(* Logix 5000 project; controller ProyectoAPMV1 vendor 1 type 14 code 156 rev 30.11; software revision 30.00 *)

TASK MainTask (continuous, watchdog 500 ms) : MainProgram

MODULES
   Local : vendor 1 type 14 code 156 (Compact 0, rev 30.11)
      DCINPUT : 1769-IQ16 (Compact 4, rev 1.1, Input RPI 20 ms)
      DCACOUTPUT : vendor 1 type 7 code 86 (Compact 5, rev 2.1, Output RPI 20 ms)
END_MODULES

VAR_GLOBAL   (* controller tags *)
   Bloquear_Puertas_Horno : BOOL;
   Buffer_Adhesivos : COUNTER := (PRE := 8);
   Buffer_Almacen : COUNTER := (PRE := 1000);
   Buffer_Calidad : COUNTER := (PRE := 8);
   Buffer_Corte : COUNTER := (PRE := 8);
   Buffer_CorteDINT : DINT;
   Buffer_Doblado : COUNTER := (PRE := 8);
   Buffer_Embalaje : COUNTER := (PRE := 100);
   Buffer_Horneado : COUNTER;
   Buffer_Pintado : COUNTER := (PRE := 100);
   Buffer_Pulido : COUNTER := (PRE := 8);
   C0 : BOOL;
   C10 : BOOL;
   C30 : BOOL;
   Contador_Calidad : COUNTER := (PRE := 100);
   E0 : BOOL;   // INICIALIZACION
   E10 : BOOL;
   E100 : BOOL;
   E110 : BOOL;
   E120 : BOOL;
   E130 : BOOL;
   E140 : BOOL;
   E150 : BOOL;
   E160 : BOOL;
   E170 : BOOL;
   E180 : BOOL;
   E190 : BOOL;
   E195 : BOOL;
   E20 : BOOL;
   E200 : BOOL;
   E210 : BOOL;
   E215 : BOOL;
   E220 : BOOL;
   E225 : BOOL;
   E230 : BOOL;
   E235 : BOOL;
   E240 : BOOL;
   E245 : BOOL;
   E250 : BOOL;
   E255 : BOOL;
   E260 : BOOL;
   E270 : BOOL;
   E280 : BOOL;
   E290 : BOOL;
   E30 : BOOL;
   E300 : BOOL;
   E310 : BOOL;
   E330 : BOOL;
   E340 : BOOL;
   E350 : BOOL;
   E360 : BOOL;
   E370 : BOOL;
   E380 : BOOL;
   E390 : BOOL;
   E40 : BOOL;
   E400 : BOOL;
   E410 : BOOL;
   E420 : BOOL;
   E430 : BOOL;
   E440 : BOOL;
   E450 : BOOL;
   E460 : BOOL;
   E50 : BOOL;
   E60 : BOOL;
   E70 : BOOL;
   E80 : BOOL;
   E90 : BOOL;
   Highlighter : BOOL;
   Lote_Piezas : DINT;
   Nro_Laminas : COUNTER := (PRE := 100);
   Parada_Pintado : BOOL;
   Piezas_Almacen : COUNTER := (PRE := 100);
   Pintado1_OK : BOOL;
   Pintado2_OK : BOOL;
   Pintado3_OK : BOOL;
   PlanseSensor2 : BOOL;
   PlanseSensor3 : BOOL;
   PlanseSensor4 : BOOL;
   Pos1ManipuladorOK : BOOL;
   Pos2ManipuladorOK : BOOL;
   Pos3ManipuladorOK : BOOL;
   Puerta_Cabina_Cerrada : BOOL;
   REINICIO_BANDERAS : BOOL;
   SCADA_Piezas : BOOL;
   Sensor_Puertas_Horno : BOOL;
   SimulationStarted : BOOL;
   Start_Adhesivos : BOOL;
   START_ALL : ALIAS FOR Local:4:I.Data.0;
   Start_Lavado : BOOL;
   Start_Pintado : BOOL;
   Start_Pulido : BOOL;
   STOP_ALL : ALIAS FOR Local:4:I.Data.1;
   Timer_Adhesivos : TIMER := (PRE := 10000);
   Timer_Alist_Adhesivos : TIMER := (PRE := 10000);
   Timer_Alist_Corte : TIMER := (PRE := 10000);
   Timer_Alist_Doblado : TIMER := (PRE := 10000);
   Timer_Alist_Embalaje : TIMER := (PRE := 10000);
   Timer_Alist_Horneado : TIMER;
   Timer_Alist_Pintado : TIMER;
   Timer_Alist_Pulido : TIMER := (PRE := 10000);
   Timer_Clasifiacion : TIMER := (PRE := 10000);
   Timer_Corte : TIMER := (PRE := 10000);
   Timer_Despacho : TIMER := (PRE := 1000);
   Timer_Doblado : TIMER := (PRE := 10000);
   Timer_Embalaje : TIMER := (PRE := 10000);
   Timer_Horneado : TIMER := (PRE := 10000);
   Timer_Lavado : TIMER := (PRE := 10000);
   Timer_Pulido : TIMER := (PRE := 10000);
   Timer_Revision_Calidad : TIMER := (PRE := 10000);
   Timer_Transp_Adhesivos : TIMER := (PRE := 10000);
   Timer_Transp_Calidad : TIMER := (PRE := 10000);
   Timer_Transp_Corte : TIMER := (PRE := 10000);
   Timer_Transp_Doblado : TIMER := (PRE := 10000);
   Timer_Transp_Embalaje : TIMER := (PRE := 10000);
   Timer_Transp_Horneado : TIMER := (PRE := 10000);
   Timer_Transp_Lavado : TIMER := (PRE := 10000);
   Timer_Transp_Pintado : TIMER;
   Timer_Transp_Pulido : TIMER := (PRE := 10000);
   Timer_Vac_Horneado : TIMER := (PRE := 1000);
END_VAR

PROGRAM MainProgram   (* main routine MainRoutine *)

ROUTINE Adhesivos   (* ladder *)
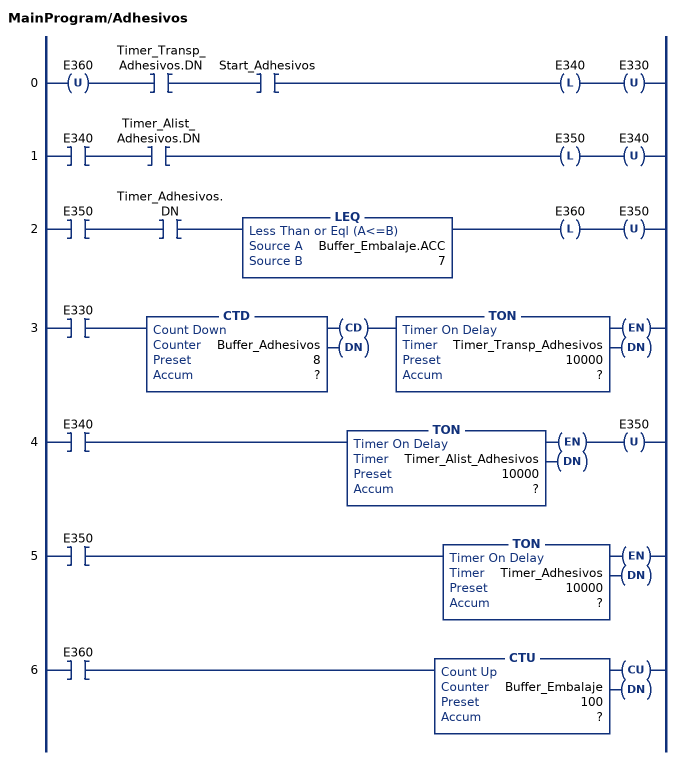
   0: OTU(E360)XIC(Timer_Transp_Adhesivos.DN)XIC(Start_Adhesivos)OTL(E340)OTU(E330);
   1: XIC(E340)XIC(Timer_Alist_Adhesivos.DN)OTL(E350)OTU(E340);
   2: XIC(E350)XIC(Timer_Adhesivos.DN)LEQ(Buffer_Embalaje.ACC,7)OTL(E360)OTU(E350);
   3: XIC(E330)CTD(Buffer_Adhesivos,?,?)TON(Timer_Transp_Adhesivos,?,?);
   4: XIC(E340)TON(Timer_Alist_Adhesivos,?,?)OTU(E350);
   5: XIC(E350)TON(Timer_Adhesivos,?,?);
   6: XIC(E360)CTU(Buffer_Embalaje,?,?);
END_ROUTINE

ROUTINE Almacen   (* ladder *)
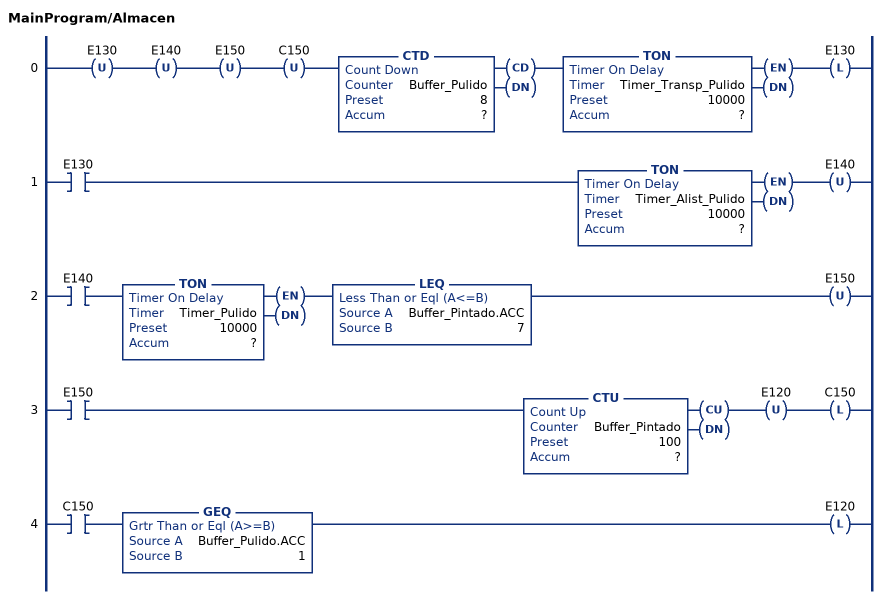
   0: OTU(E130)OTU(E140)OTU(E150)OTU(C150)CTD(Buffer_Pulido,?,?)TON(Timer_Transp_Pulido,?,?)OTL(E130);
   1: XIC(E130)TON(Timer_Alist_Pulido,?,?)OTU(E140);
   2: XIC(E140)TON(Timer_Pulido,?,?)LEQ(Buffer_Pintado.ACC,7)OTU(E150);
   3: XIC(E150)CTU(Buffer_Pintado,?,?)OTU(E120)OTL(C150);
   4: XIC(C150)GEQ(Buffer_Pulido.ACC,1)OTL(E120);
END_ROUTINE

ROUTINE Calidad   (* ladder *)
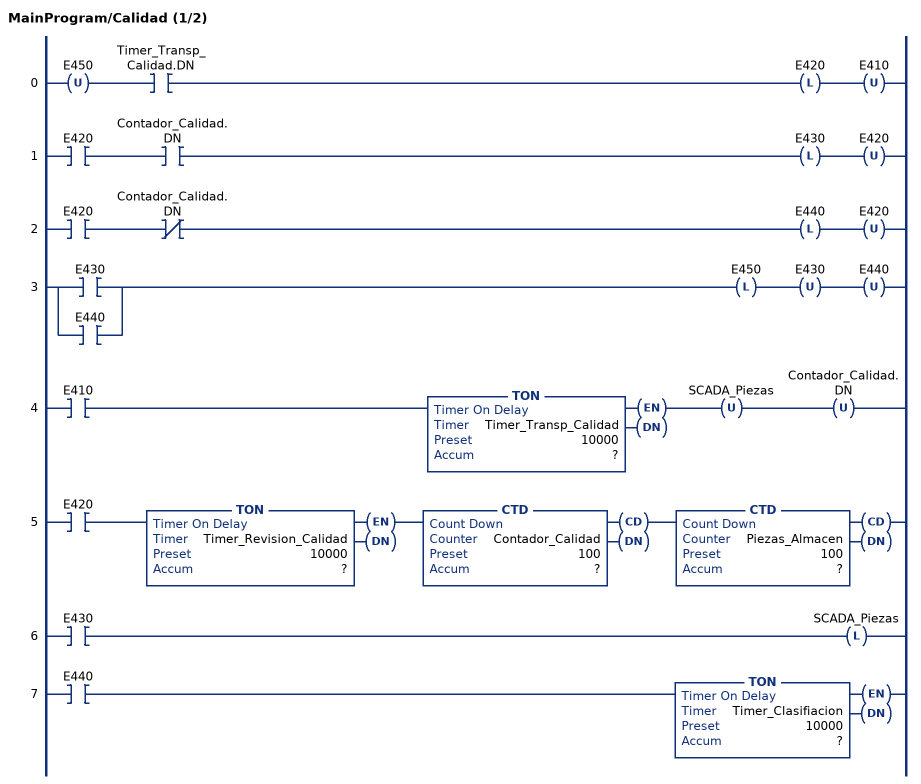
   0: OTU(E450)XIC(Timer_Transp_Calidad.DN)OTL(E420)OTU(E410);
   1: XIC(E420)XIC(Contador_Calidad.DN)OTL(E430)OTU(E420);
   2: XIC(E420)XIO(Contador_Calidad.DN)OTL(E440)OTU(E420);
   3: [XIC(E430) ,XIC(E440) ]OTL(E450)OTU(E430)OTU(E440);
   4: XIC(E410)TON(Timer_Transp_Calidad,?,?)OTU(SCADA_Piezas)OTU(Contador_Calidad.DN);
   5: XIC(E420)TON(Timer_Revision_Calidad,?,?)CTD(Contador_Calidad,?,?)CTD(Piezas_Almacen,?,?);
   6: XIC(E430)OTL(SCADA_Piezas);
   7: XIC(E440)TON(Timer_Clasifiacion,?,?);
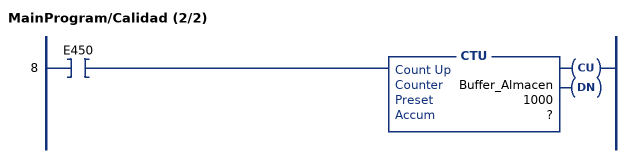
   8: XIC(E450)CTU(Buffer_Almacen,?,?);
END_ROUTINE

ROUTINE Corte_Laminas   (* ladder *)
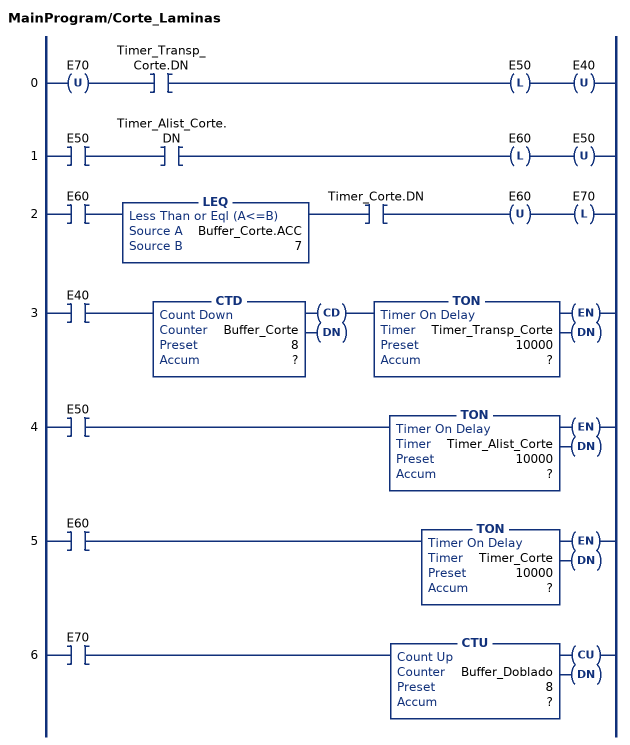
   0: OTU(E70)XIC(Timer_Transp_Corte.DN)OTL(E50)OTU(E40);
   1: XIC(E50)XIC(Timer_Alist_Corte.DN)OTL(E60)OTU(E50);
   2: XIC(E60)LEQ(Buffer_Corte.ACC,7)XIC(Timer_Corte.DN)OTU(E60)OTL(E70);
   3: XIC(E40)CTD(Buffer_Corte,?,?)TON(Timer_Transp_Corte,?,?);
   4: XIC(E50)TON(Timer_Alist_Corte,?,?);
   5: XIC(E60)TON(Timer_Corte,?,?);
   6: XIC(E70)CTU(Buffer_Doblado,?,?);
END_ROUTINE

ROUTINE Doblado_Laminas   (* ladder *)
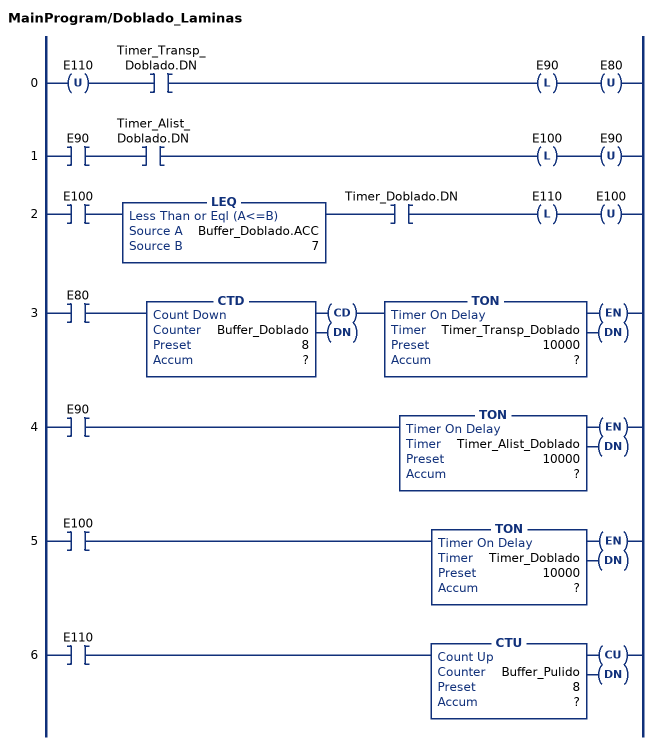
   0: OTU(E110)XIC(Timer_Transp_Doblado.DN)OTL(E90)OTU(E80);
   1: XIC(E90)XIC(Timer_Alist_Doblado.DN)OTL(E100)OTU(E90);
   2: XIC(E100)LEQ(Buffer_Doblado.ACC,7)XIC(Timer_Doblado.DN)OTL(E110)OTU(E100);
   3: XIC(E80)CTD(Buffer_Doblado,?,?)TON(Timer_Transp_Doblado,?,?);
   4: XIC(E90)TON(Timer_Alist_Doblado,?,?);
   5: XIC(E100)TON(Timer_Doblado,?,?);
   6: XIC(E110)CTU(Buffer_Pulido,?,?);
END_ROUTINE

ROUTINE Embalaje   (* ladder *)
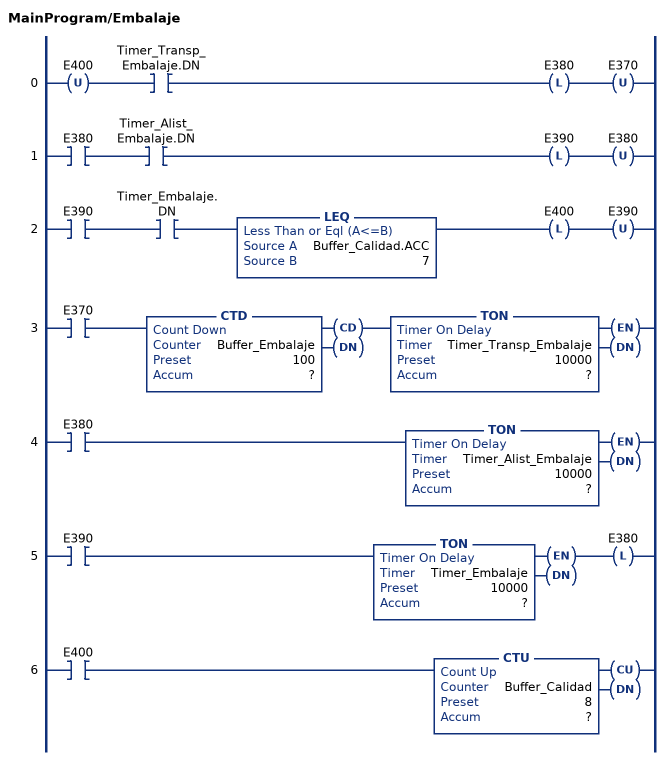
   0: OTU(E400)XIC(Timer_Transp_Embalaje.DN)OTL(E380)OTU(E370);
   1: XIC(E380)XIC(Timer_Alist_Embalaje.DN)OTL(E390)OTU(E380);
   2: XIC(E390)XIC(Timer_Embalaje.DN)LEQ(Buffer_Calidad.ACC,7)OTL(E400)OTU(E390);
   3: XIC(E370)CTD(Buffer_Embalaje,?,?)TON(Timer_Transp_Embalaje,?,?);
   4: XIC(E380)TON(Timer_Alist_Embalaje,?,?);
   5: XIC(E390)TON(Timer_Embalaje,?,?)OTL(E380);
   6: XIC(E400)CTU(Buffer_Calidad,?,?);
END_ROUTINE

ROUTINE Horneado_Piezas   (* ladder *)
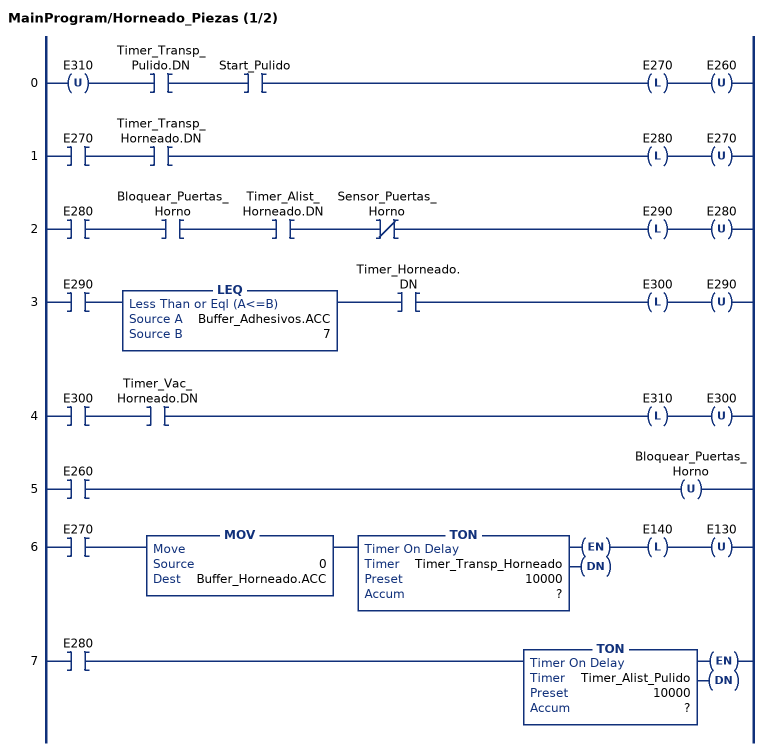
   0: OTU(E310)XIC(Timer_Transp_Pulido.DN)XIC(Start_Pulido)OTL(E270)OTU(E260);
   1: XIC(E270)XIC(Timer_Transp_Horneado.DN)OTL(E280)OTU(E270);
   2: XIC(E280)XIC(Bloquear_Puertas_Horno)XIC(Timer_Alist_Horneado.DN)XIO(Sensor_Puertas_Horno)OTL(E290)OTU(E280);
   3: XIC(E290)LEQ(Buffer_Adhesivos.ACC,7)XIC(Timer_Horneado.DN)OTL(E300)OTU(E290);
   4: XIC(E300)XIC(Timer_Vac_Horneado.DN)OTL(E310)OTU(E300);
   5: XIC(E260)OTU(Bloquear_Puertas_Horno);
   6: XIC(E270)MOV(0,Buffer_Horneado.ACC)TON(Timer_Transp_Horneado,?,?)OTL(E140)OTU(E130);
   7: XIC(E280)TON(Timer_Alist_Pulido,?,?);
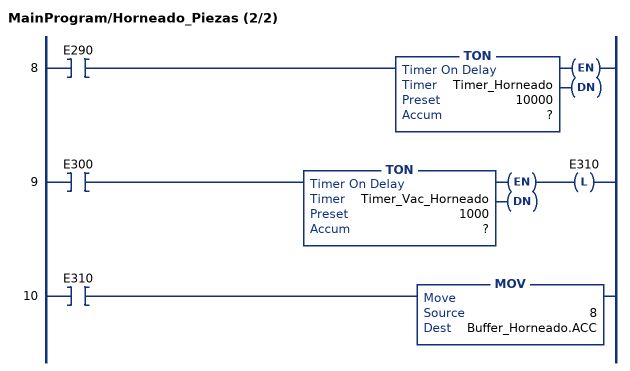
   8: XIC(E290)TON(Timer_Horneado,?,?);
   9: XIC(E300)TON(Timer_Vac_Horneado,?,?)OTL(E310);
   10: XIC(E310)MOV(8,Buffer_Horneado.ACC);
END_ROUTINE

ROUTINE Lavado_Laminas   (* ladder *)
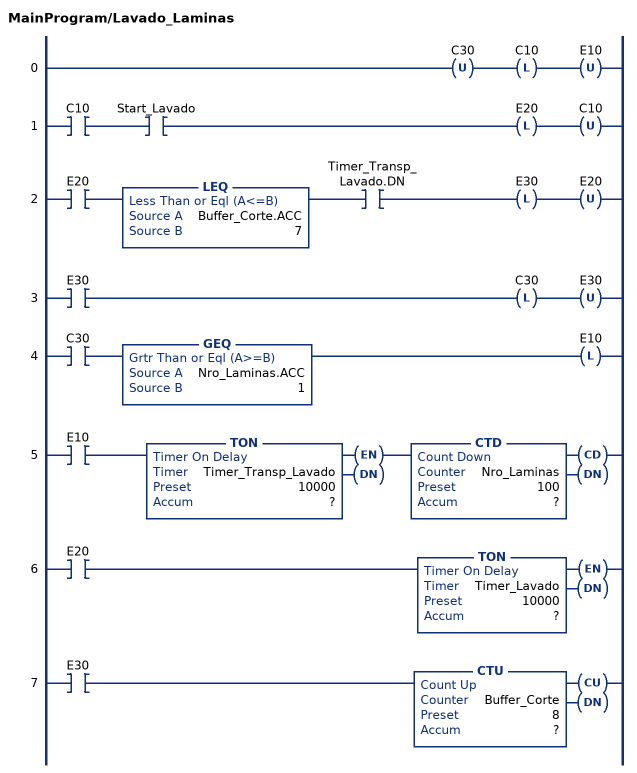
   0: OTU(C30)OTL(C10)OTU(E10);
   1: XIC(C10)XIC(Start_Lavado)OTL(E20)OTU(C10);
   2: XIC(E20)LEQ(Buffer_Corte.ACC,7)XIC(Timer_Transp_Lavado.DN)OTL(E30)OTU(E20);
   3: XIC(E30)OTL(C30)OTU(E30);
   4: XIC(C30)GEQ(Nro_Laminas.ACC,1)OTL(E10);
   5: XIC(E10)TON(Timer_Transp_Lavado,?,?)CTD(Nro_Laminas,?,?);
   6: XIC(E20)TON(Timer_Lavado,?,?);
   7: XIC(E30)CTU(Buffer_Corte,?,?);
END_ROUTINE

ROUTINE MainRoutine   (* ladder *)
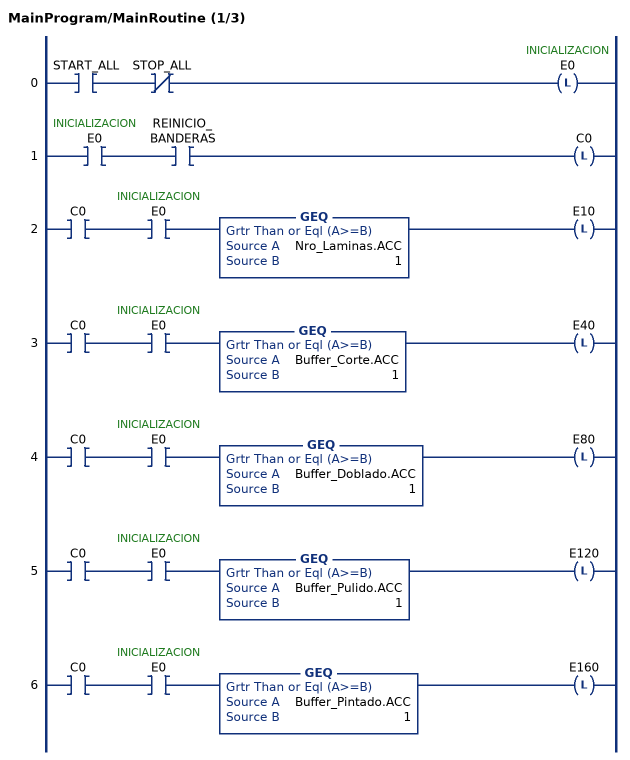
   0: XIC(START_ALL)XIO(STOP_ALL)OTL(E0);
   1: XIC(E0)XIC(REINICIO_BANDERAS)OTL(C0);
   2: XIC(C0)XIC(E0)GEQ(Nro_Laminas.ACC,1)OTL(E10);
   3: XIC(C0)XIC(E0)GEQ(Buffer_Corte.ACC,1)OTL(E40);
   4: XIC(C0)XIC(E0)GEQ(Buffer_Doblado.ACC,1)OTL(E80);
   5: XIC(C0)XIC(E0)GEQ(Buffer_Pulido.ACC,1)OTL(E120);
   6: XIC(C0)XIC(E0)GEQ(Buffer_Pintado.ACC,1)OTL(E160);
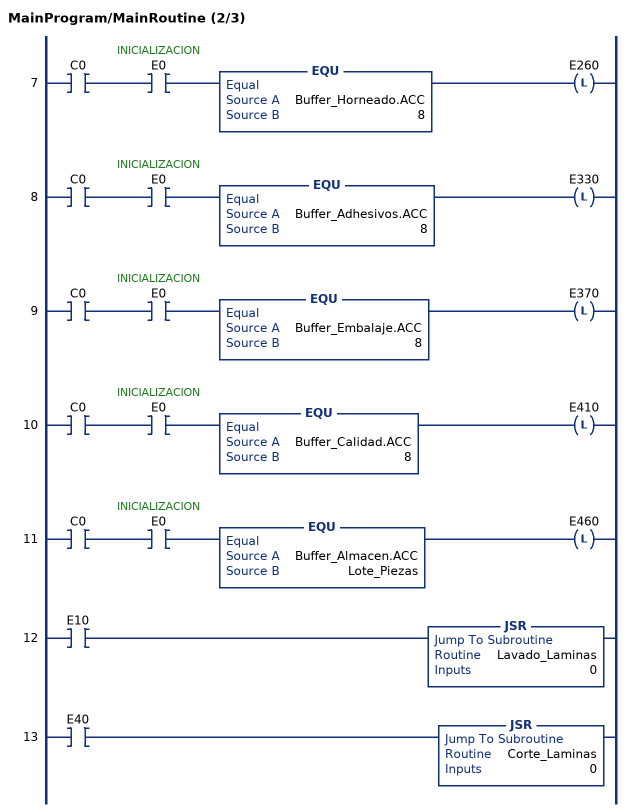
   7: XIC(C0)XIC(E0)EQU(Buffer_Horneado.ACC,8)OTL(E260);
   8: XIC(C0)XIC(E0)EQU(Buffer_Adhesivos.ACC,8)OTL(E330);
   9: XIC(C0)XIC(E0)EQU(Buffer_Embalaje.ACC,8)OTL(E370);
   10: XIC(C0)XIC(E0)EQU(Buffer_Calidad.ACC,8)OTL(E410);
   11: XIC(C0)XIC(E0)EQU(Buffer_Almacen.ACC,Lote_Piezas)OTL(E460);
   12: XIC(E10)JSR(Lavado_Laminas,0);
   13: XIC(E40)JSR(Corte_Laminas,0);
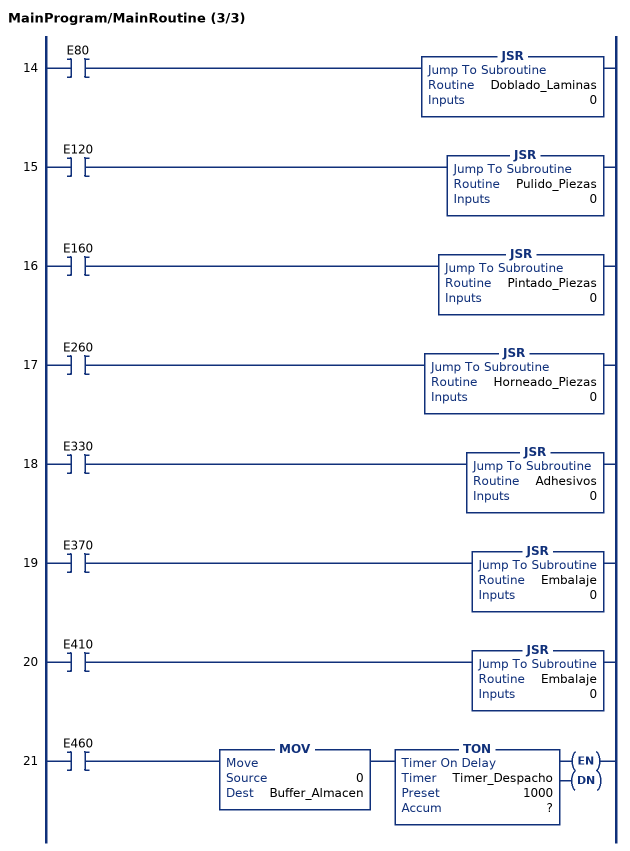
   14: XIC(E80)JSR(Doblado_Laminas,0);
   15: XIC(E120)JSR(Pulido_Piezas,0);
   16: XIC(E160)JSR(Pintado_Piezas,0);
   17: XIC(E260)JSR(Horneado_Piezas,0);
   18: XIC(E330)JSR(Adhesivos,0);
   19: XIC(E370)JSR(Embalaje,0);
   20: XIC(E410)JSR(Embalaje,0);
   21: XIC(E460)MOV(0,Buffer_Almacen)TON(Timer_Despacho,?,?);
END_ROUTINE

ROUTINE Pintado_Piezas   (* ladder *)
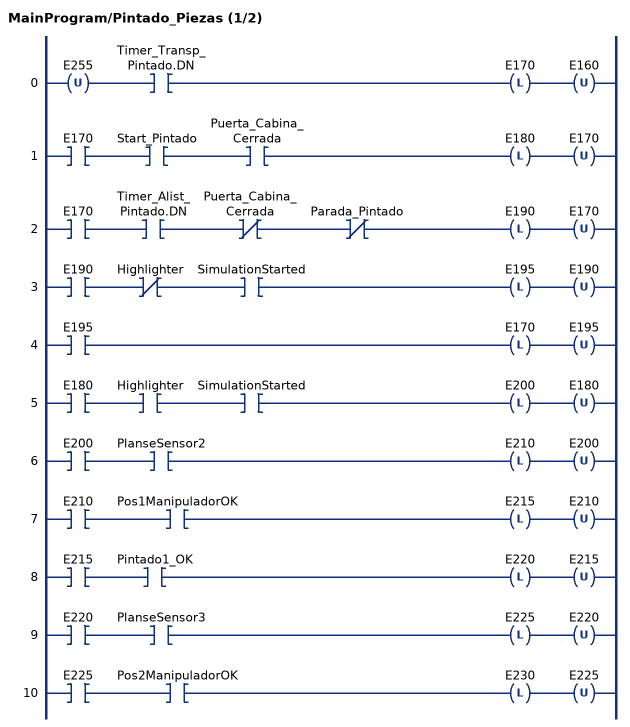
   0: OTU(E255)XIC(Timer_Transp_Pintado.DN)OTL(E170)OTU(E160);
   1: XIC(E170)XIC(Start_Pintado)XIC(Puerta_Cabina_Cerrada)OTL(E180)OTU(E170);
   2: XIC(E170)XIC(Timer_Alist_Pintado.DN)XIO(Puerta_Cabina_Cerrada)XIO(Parada_Pintado)OTL(E190)OTU(E170);
   3: XIC(E190)XIO(Highlighter)XIC(SimulationStarted)OTL(E195)OTU(E190);
   4: XIC(E195)OTL(E170)OTU(E195);
   5: XIC(E180)XIC(Highlighter)XIC(SimulationStarted)OTL(E200)OTU(E180);
   6: XIC(E200)XIC(PlanseSensor2)OTL(E210)OTU(E200);
   7: XIC(E210)XIC(Pos1ManipuladorOK)OTL(E215)OTU(E210);
   8: XIC(E215)XIC(Pintado1_OK)OTL(E220)OTU(E215);
   9: XIC(E220)XIC(PlanseSensor3)OTL(E225)OTU(E220);
   10: XIC(E225)XIC(Pos2ManipuladorOK)OTL(E230)OTU(E225);
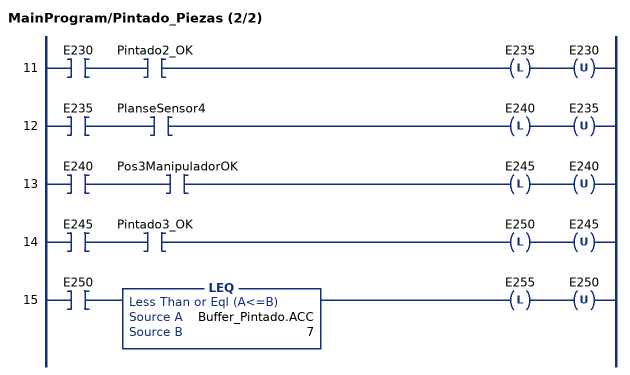
   11: XIC(E230)XIC(Pintado2_OK)OTL(E235)OTU(E230);
   12: XIC(E235)XIC(PlanseSensor4)OTL(E240)OTU(E235);
   13: XIC(E240)XIC(Pos3ManipuladorOK)OTL(E245)OTU(E240);
   14: XIC(E245)XIC(Pintado3_OK)OTL(E250)OTU(E245);
   15: XIC(E250)LEQ(Buffer_Pintado.ACC,7)OTL(E255)OTU(E250);
END_ROUTINE

ROUTINE Pulido_Piezas   (* ladder *)
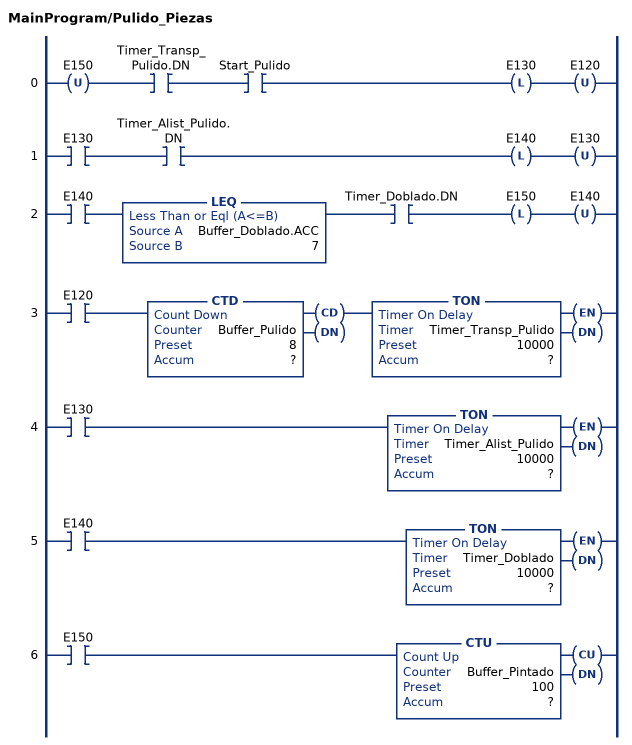
   0: OTU(E150)XIC(Timer_Transp_Pulido.DN)XIC(Start_Pulido)OTL(E130)OTU(E120);
   1: XIC(E130)XIC(Timer_Alist_Pulido.DN)OTL(E140)OTU(E130);
   2: XIC(E140)LEQ(Buffer_Doblado.ACC,7)XIC(Timer_Doblado.DN)OTL(E150)OTU(E140);
   3: XIC(E120)CTD(Buffer_Pulido,?,?)TON(Timer_Transp_Pulido,?,?);
   4: XIC(E130)TON(Timer_Alist_Pulido,?,?);
   5: XIC(E140)TON(Timer_Doblado,?,?);
   6: XIC(E150)CTU(Buffer_Pintado,?,?);
END_ROUTINE
END_PROGRAM
